Fanuc KAREL source: wutool.kl

PROGRAM wutool
%NOLOCKGROUP
VAR
  p : POSITION
  q : POSITION
  i : INTEGER
  r : REAL
BEGIN
  WITH $UTOOL = p MOVE TO p
END wutool
